FUNCTION_BLOCK AdjustableSizeReplyRpcHandler IMPLEMENTS I_SynchronousRpcHandler
VAR
END_VAR

METHOD Handle
VAR_INPUT
	Parameters : I_Deserializer;
	Response : I_SynchronousRpcResponse;
END_VAR
VAR
	deserializerFeedback : DeserializerFeedback;
	size : UDINT;
	pBytes : POINTER TO BYTE;
	currentPos : POINTER TO BYTE;
	i : UDINT;
	count : BYTE;
END_VAR
IF NOT Parameters.TryGetKeyUdint('Size', size, deserializerFeedback) THEN
	Response.RejectWithMessage('Missing Size parameter');
	RETURN;
END_IF

IF size = 0 THEN 
	Response.CompleteWithNull();
END_IF

pBytes := __NEW(BYTE, size);
FOR i := 0 TO size -1 DO
	currentPos := pBytes + i;
	currentPos^ := count;
	count := count + 1;
END_FOR

Response.CompleteWithBytesAsHex(pBytes, UDINT_TO_DINT(size));

__Delete(pBytes);
END_METHOD

END_FUNCTION_BLOCK

(* stored: Version 1.1.0.1, ProductVersion 3.1.4024.13
   POU AdjustableSizeReplyRpcHandler: Id {9299e15a-1853-4d5c-887c-44fb5a606abe}, SpecialFunc None
   Method Handle: Id {9f2bbb3b-e3e7-4379-9b54-5579b5c73f06} *)
